// TIA Portal V18 export
VAR_GLOBAL   // PLC tag table "MES_TotalResult"
END_VAR
VAR_GLOBAL CONSTANT   // user constants
   MES_ProcessResultNG_Press : Int := 2;
   MES_ProcessResultOK : Int := 1;
   MES_ProcessResultIDIE : Int := 0;
END_VAR
